(* PLC project Cell Example , CTH FIX1 1.0, author CTH SS2 *)
(* stored: companyURL www.chalmers.se, creationDateTime 2008-03-19T20:31:26, version 1.0, modificationDateTime 2008-05-13T18:21:07, organization SS2, language en-US *)

TYPE BinaryPositions : ();
END_TYPE

FUNCTION ADD_E : INT
  VAR_INPUT
    Enable : BOOL := FALSE;
    IN1 : INT := 0;
    IN2 : INT := 0;
  END_VAR
  VAR_OUTPUT
    EnableO : BOOL := FALSE;
  END_VAR

(* LD diagram, written out as Structured Text *)
END_FUNCTION

FUNCTION DEC_E : INT
  VAR_INPUT
    Enable : BOOL;
  END_VAR
  VAR_OUTPUT
    EnableO : BOOL;
  END_VAR

(* LD diagram, written out as Structured Text *)
END_FUNCTION

FUNCTION MOVE_E : STRING
  VAR_INPUT
    Enable : BOOL := FALSE;
    IN : STRING;
  END_VAR
  VAR_OUTPUT
    EnableO : BOOL := FALSE;
  END_VAR

(* LD diagram, written out as Structured Text *)
END_FUNCTION

FUNCTION_BLOCK test4
  VAR_INPUT
    i1 : BOOL := FALSE;
  END_VAR
  VAR_OUTPUT
    o1 : BOOL := TRUE;
  END_VAR

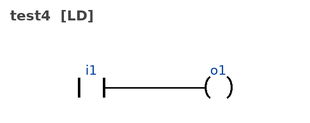
(* LD diagram, written out as Structured Text *)
o1 := i1;
END_FUNCTION_BLOCK

FUNCTION_BLOCK test2
  VAR_INPUT
    i : BOOL;
  END_VAR
  VAR_OUTPUT
    o : BOOL;
  END_VAR
  VAR
    internal1 : test4;
  END_VAR

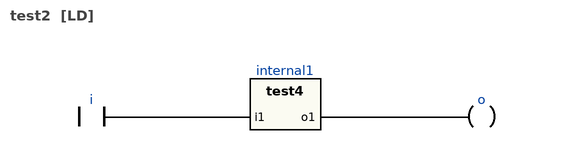
(* LD diagram, written out as Structured Text *)
internal1(i1 := i);
o := internal1.o1;
END_FUNCTION_BLOCK

FUNCTION_BLOCK test5
  VAR_INPUT
    in : BOOL;
  END_VAR
  VAR_OUTPUT
    ut : BOOL;
  END_VAR

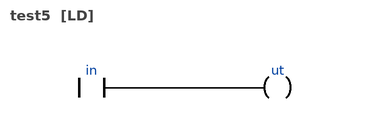
(* LD diagram, written out as Structured Text *)
ut := in;
END_FUNCTION_BLOCK

FUNCTION_BLOCK test3
  VAR_INPUT
    in1 : BOOL;
  END_VAR
  VAR_OUTPUT
    ut1 : BOOL;
  END_VAR
  VAR
    internal1 : test4;
    internal2 : test5;
  END_VAR

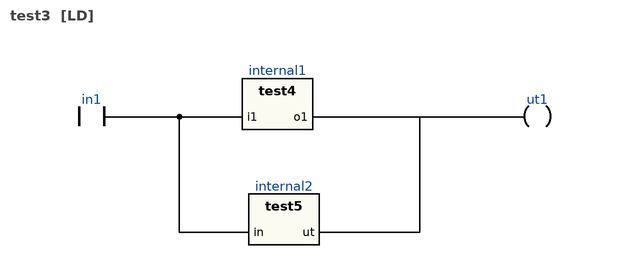
(* LD diagram, written out as Structured Text *)
internal1(i1 := in1);
internal2(in := in1);
ut1 := internal1.o1 OR internal2.ut;
END_FUNCTION_BLOCK

FUNCTION_BLOCK TestFB
  VAR_INPUT
    IN1 : BOOL := FALSE;
    IN2 : INT := 0;
    IN3 : BOOL := FALSE;
  END_VAR
  VAR_OUTPUT
    OUT1 : BOOL := FALSE;
    OUT2 : BOOL := FALSE;
    OUT3 : BOOL := FALSE;
    OUT4 : INT := 0;
  END_VAR
  VAR
    internal1 : test2;
    internal2 : test3;
  END_VAR

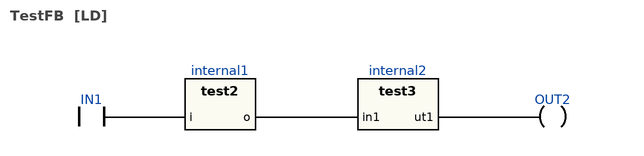
(* LD diagram, written out as Structured Text *)
internal1(i := IN1);
internal2(in1 := internal1.o);
OUT2 := internal2.ut1;
END_FUNCTION_BLOCK

FUNCTION_BLOCK RAC
  VAR_INPUT
    IN1 : BOOL := FALSE;
  END_VAR
  VAR_OUTPUT
    OUT : BOOL := FALSE;
  END_VAR
  VAR_INPUT
    IN2 : BOOL := TRUE;
  END_VAR
  VAR
    Var3 : BOOL := TRUE;
    IN4 : INT := 5;
  END_VAR
  VAR_OUTPUT
    State : STRING := 'Undefined';
  END_VAR
  VAR
    timer : TON;
    passedTime : TIME := 20;
    test : TestFB;
  END_VAR
  VAR_OUTPUT
    OUT2 : BOOL := TRUE;
  END_VAR
  VAR  (* added by the conversion: wires and edge detectors of the diagram *)
    _ADD_E24_ : ANY;
    _ADD_E24_OUT : INT;
    _MOVE_E26_ : ANY;
    _MOVE_E26_OUT : STRING;
    _DEC_E34_ : ANY;
    _DEC_E34_OUT : INT;
  END_VAR

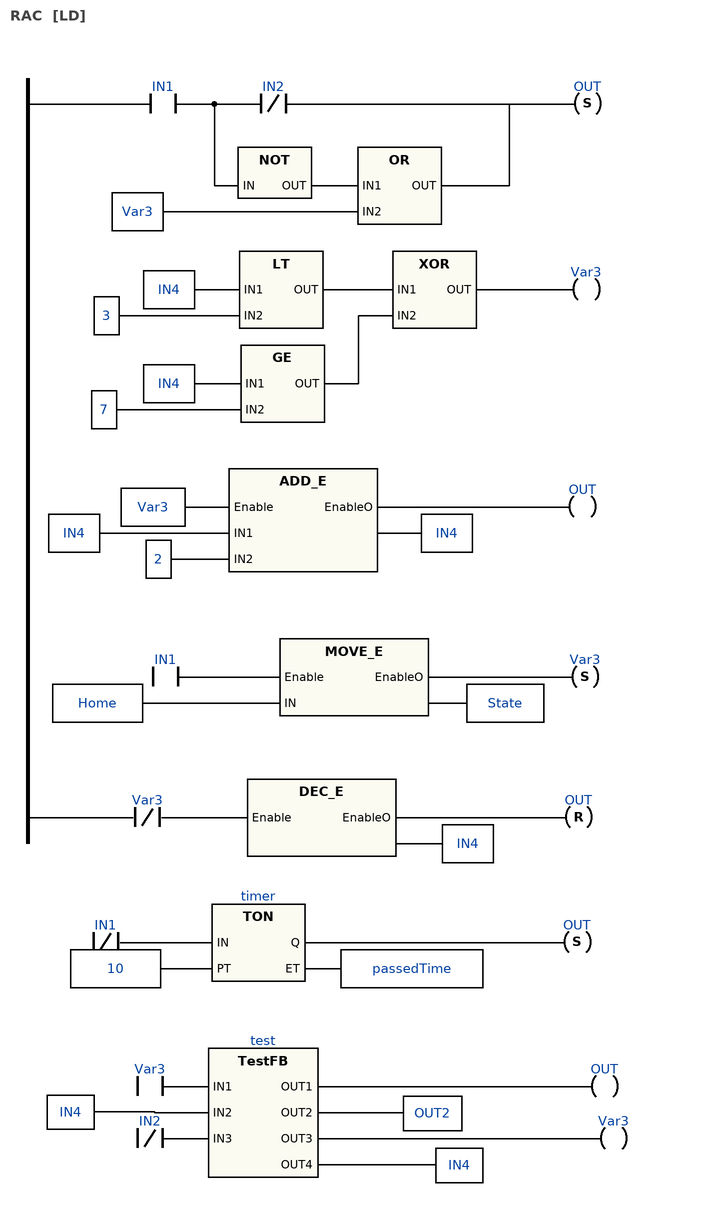
(* LD diagram, written out as Structured Text *)
IF IN1 AND NOT IN2 OR NOT IN1 OR Var3 THEN OUT := TRUE; END_IF;
Var3 := IN4 < 3 XOR IN4 >= 7;
_ADD_E24_OUT := ADD_E(Enable := Var3, IN1 := IN4, IN2 := 2,  => _ADD_E24_);
OUT := _ADD_E24_OUT;
IN4 := _ADD_E24_OUT;
_MOVE_E26_OUT := MOVE_E(Enable := IN1, IN := Home,  => _MOVE_E26_);
IF _MOVE_E26_OUT THEN Var3 := TRUE; END_IF;
State := _MOVE_E26_OUT;
_DEC_E34_OUT := DEC_E(Enable := NOT Var3,  => _DEC_E34_);
IF _DEC_E34_OUT THEN OUT := FALSE; END_IF;
IN4 := _DEC_E34_OUT;
timer(IN := NOT IN1, PT := 10);
IF timer.Q THEN OUT := TRUE; END_IF;
passedTime := timer.ET;
test(IN1 := Var3, IN2 := IN4, IN3 := NOT IN2);
OUT := test.OUT1;
OUT2 := test.OUT2;
Var3 := test.OUT3;
IN4 := test.OUT4;
END_FUNCTION_BLOCK

CONFIGURATION ExampleCell
END_CONFIGURATION
